Universal Robots PolyScope program: Depl90.urp

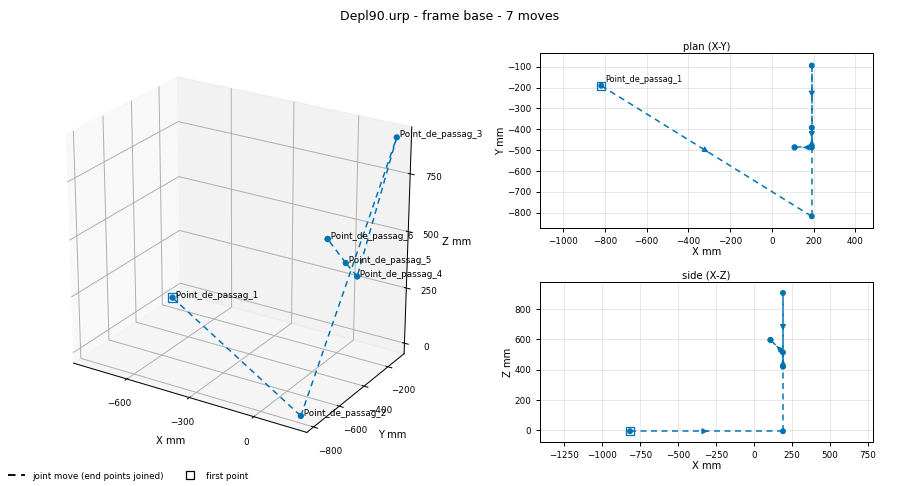
[picture p0: tool path of Depl90.urp in frame base, 7 of 7 moves have a stored position in this frame; points joined in program order, loops and branches not executed]
ProgramRoot directory=/home/dominique/ursim-1.6_UR5/programs; kinematics=(a=[0, -0.425, -0.39225, 0, 0, 0], d=[0.08916, 0, 0, 0.10915, 0.09465, 0.0823], alpha=[1.5708, 0, 0, 1.5708, -1.5708, 0], deltaTheta=[0, 0, 0, 0, 0, 0], status=notInitialized); name=Depl90; programVersion=(project__name=PolyScope, major__version=1, minor__version=6, svn__revision=8725, build__date=Jul 31 2012, 11:04:51); robotEnvironmentFileName=default
  MainProgram cartesianAcceleration=1.2; cartesianSpeed=0.25; jointAcceleration=1.3962634015954636; jointSpeed=1.0471975511965976; moveAsFastAsPossible=true; sharedProcessMoveBlendRadius=0.025; featureReference=(installationNameReference=Base); motionType=JOINT_SPACE
    Move cartesianAcceleration=1.2; cartesianSpeed=0.25; jointAcceleration=1.3962634015954636; jointSpeed=1.0471975511965976; moveAsFastAsPossible=true; sharedProcessMoveBlendRadius=0.025; featureReference=(installationNameReference=Base); motionType=JOINT_SPACE
      Waypoint blendRadius=0.05; cartesianAcceleration=1.2; cartesianSpeed=0.25; jointAcceleration=1.3962634015954636; jointSpeed=1.0471975511965976; nextMotionTime=2.0; stoppoint=true; useSharedBlendParameter=true; useSharedParameters=true; position=TCP in base x=-817.25 y=-191.45 z=-5.491 mm, rx=1.5708 ry=0 rz=0 rad; joints [0, 0, 0, 0, 0, 0] deg; positionType=FIXED_POSITION; waypointPoseInFeatureCoordinates=(pos=(x=-0.8172499999999999, y=-0.1914499999611738, z=-0.005491000039267544), rot=(x=1.570796327, y=-1.277447271408914E-15, z=3.1862404642400186E-16)); name=Point_de_passag_1
      Wait analogComparison=0; analogInputRange=0; analogValue=0.0; digitalValue=0; selectedAnalogSensor=-1; selectedDigitalSensor=-1; waitTime=1.0; type=TIMER_WAIT
    Move cartesianAcceleration=1.2; cartesianSpeed=0.25; jointAcceleration=1.3962634015954636; jointSpeed=1.0471975511965976; moveAsFastAsPossible=true; sharedProcessMoveBlendRadius=0.025; featureReference=(installationNameReference=Base); motionType=JOINT_SPACE
      Waypoint blendRadius=0.05; cartesianAcceleration=1.2; cartesianSpeed=0.25; jointAcceleration=1.3962634015954636; jointSpeed=1.0471975511965976; nextMotionTime=2.0; stoppoint=true; useSharedBlendParameter=true; useSharedParameters=true; position=TCP in base x=191.45 y=-817.25 z=-5.491 mm, rx=1.2092 ry=1.2092 rz=1.2092 rad; joints [90, 0, 0, 0, 0, 0] deg; positionType=FIXED_POSITION; waypointPoseInFeatureCoordinates=(pos=(x=0.19144999996117368, y=-0.81725, z=-0.005491000039267544), rot=(x=1.2091995763071843, y=1.2091995763071826, z=1.209199576059173)); name=Point_de_passag_2
      Waypoint blendRadius=0.05; cartesianAcceleration=1.2; cartesianSpeed=0.25; jointAcceleration=1.3962634015954636; jointSpeed=1.0471975511965976; nextMotionTime=2.0; stoppoint=true; useSharedBlendParameter=true; useSharedParameters=true; position=TCP in base x=191.45 y=-94.65 z=906.409 mm, rx=0 ry=1.5708 rz=0 rad; joints [90, -90, 0, 0, 0, 0] deg; positionType=FIXED_POSITION; waypointPoseInFeatureCoordinates=(pos=(x=0.1914500001482077, y=-0.0946500000000019, z=0.9064089999607328), rot=(x=1.8458863867508093E-15, y=1.5707963269999994, z=1.4009191784961424E-15)); name=Point_de_passag_3
      Waypoint blendRadius=0.05; cartesianAcceleration=1.2; cartesianSpeed=0.25; jointAcceleration=1.3962634015954636; jointSpeed=1.0471975511965976; nextMotionTime=2.0; stoppoint=true; useSharedBlendParameter=true; useSharedParameters=true; position=TCP in base x=191.45 y=-392.25 z=419.509 mm, rx=1.2092 ry=1.2092 rz=1.2092 rad; joints [90, -90, 90, 0, 0, 0] deg; positionType=FIXED_POSITION; waypointPoseInFeatureCoordinates=(pos=(x=0.19145000004834276, y=-0.392250000000001, z=0.4195089999607324), rot=(x=1.209199576307185, y=1.2091995763071821, z=1.2091995760591734)); name=Point_de_passag_4
      Waypoint blendRadius=0.05; cartesianAcceleration=1.2; cartesianSpeed=0.25; jointAcceleration=1.3962634015954636; jointSpeed=1.0471975511965976; nextMotionTime=2.0; stoppoint=true; useSharedBlendParameter=true; useSharedParameters=true; position=TCP in base x=191.45 y=-486.9 z=514.159 mm, rx=0 ry=1.5708 rz=0 rad; joints [90, -90, 90, -90, 0, 0] deg; positionType=FIXED_POSITION; waypointPoseInFeatureCoordinates=(pos=(x=0.19145000006775575, y=-0.4869000000000011, z=0.5141589999607317), rot=(x=3.927026672455434E-15, y=1.5707963269999994, z=3.482059463774424E-15)); name=Point_de_passag_5
      Waypoint blendRadius=0.05; cartesianAcceleration=1.2; cartesianSpeed=0.25; jointAcceleration=1.3962634015954636; jointSpeed=1.0471975511965976; nextMotionTime=2.0; stoppoint=true; useSharedBlendParameter=true; useSharedParameters=true; position=TCP in base x=109.15 y=-486.9 z=596.459 mm, rx=0 ry=0 rz=0 rad; joints [90, -90, 90, -90, 90, 0] deg; positionType=FIXED_POSITION; waypointPoseInFeatureCoordinates=(pos=(x=0.10915000008463584, y=-0.4868999999831215, z=0.5964589999776116), rot=(x=0.0, y=0.0, z=0.0)); name=Point_de_passag_6
      Waypoint blendRadius=0.05; cartesianAcceleration=1.2; cartesianSpeed=0.25; jointAcceleration=1.3962634015954636; jointSpeed=1.0471975511965976; nextMotionTime=2.0; stoppoint=true; useSharedBlendParameter=true; useSharedParameters=true; position=TCP in base x=109.15 y=-486.9 z=596.459 mm, rx=0 ry=0 rz=1.5708 rad; joints [90, -90, 90, -90, 90, 90] deg; positionType=FIXED_POSITION; waypointPoseInFeatureCoordinates=(pos=(x=0.10915000008463582, y=-0.4868999999831215, z=0.5964589999776116), rot=(x=4.107229131184617E-15, y=3.221723986770376E-10, z=1.5707963265897928)); name=Point_de_passag_7
